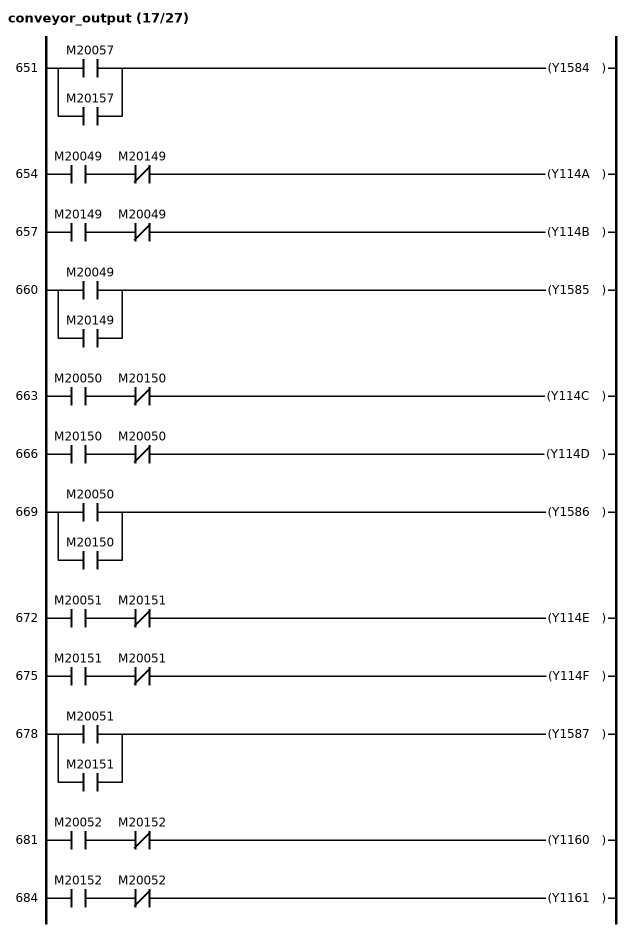
[picture p144: ladder of conveyor_output, rungs at steps 651 to 684]
651   LD      M20057
      OR      M20157
      OUT     Y1584
654   LD      M20049
      ANI     M20149
      OUT     Y114A
657   LD      M20149
      ANI     M20049
      OUT     Y114B
660   LD      M20049
      OR      M20149
      OUT     Y1585
663   LD      M20050
      ANI     M20150
      OUT     Y114C
666   LD      M20150
      ANI     M20050
      OUT     Y114D
669   LD      M20050
      OR      M20150
      OUT     Y1586
672   LD      M20051
      ANI     M20151
      OUT     Y114E
675   LD      M20151
      ANI     M20051
      OUT     Y114F
678   LD      M20051
      OR      M20151
      OUT     Y1587
681   LD      M20052
      ANI     M20152
      OUT     Y1160
684   LD      M20152
      ANI     M20052
      OUT     Y1161
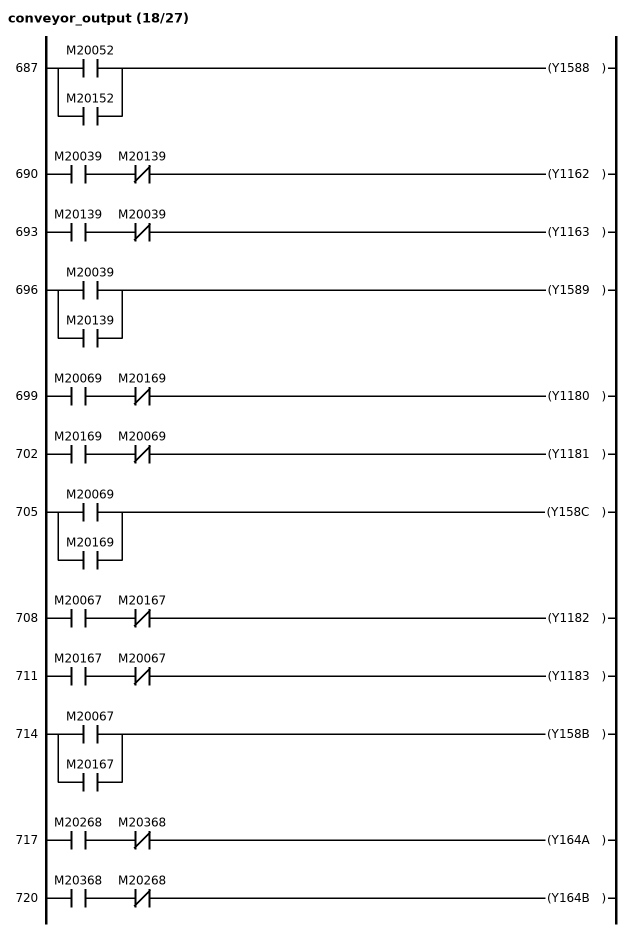
687   LD      M20052
      OR      M20152
      OUT     Y1588
690   LD      M20039
      ANI     M20139
      OUT     Y1162
693   LD      M20139
      ANI     M20039
      OUT     Y1163
696   LD      M20039
      OR      M20139
      OUT     Y1589
699   LD      M20069
      ANI     M20169
      OUT     Y1180
702   LD      M20169
      ANI     M20069
      OUT     Y1181
705   LD      M20069
      OR      M20169
      OUT     Y158C
708   LD      M20067
      ANI     M20167
      OUT     Y1182
711   LD      M20167
      ANI     M20067
      OUT     Y1183
714   LD      M20067
      OR      M20167
      OUT     Y158B
717   LD      M20268
      ANI     M20368
      OUT     Y164A
720   LD      M20368
      ANI     M20268
      OUT     Y164B
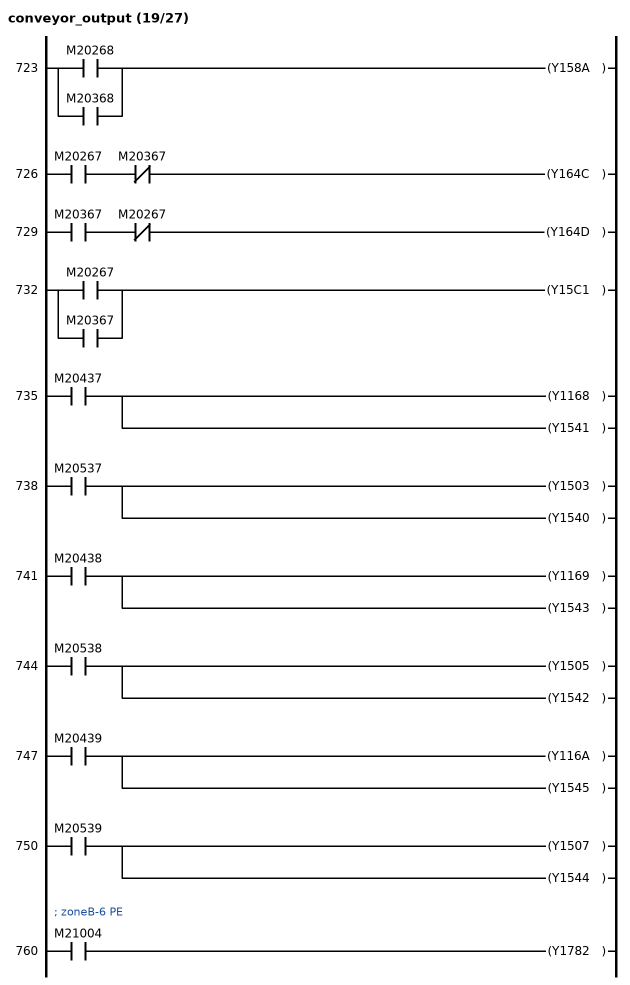
723   LD      M20268
      OR      M20368
      OUT     Y158A
726   LD      M20267
      ANI     M20367
      OUT     Y164C
729   LD      M20367
      ANI     M20267
      OUT     Y164D
732   LD      M20267
      OR      M20367
      OUT     Y15C1
735   LD      M20437
      OUT     Y1168
      OUT     Y1541
738   LD      M20537
      OUT     Y1503
      OUT     Y1540
741   LD      M20438
      OUT     Y1169
      OUT     Y1543
744   LD      M20538
      OUT     Y1505
      OUT     Y1542
747   LD      M20439
      OUT     Y116A
      OUT     Y1545
750   LD      M20539
      OUT     Y1507
      OUT     Y1544
; zoneB-6 PE
760   LD      M21004
      OUT     Y1782
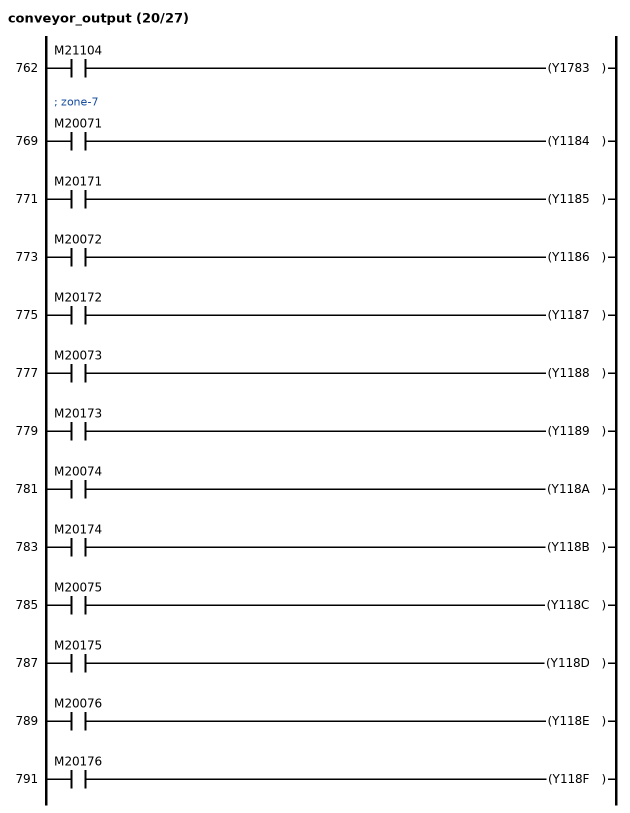
762   LD      M21104
      OUT     Y1783
; zone-7
769   LD      M20071
      OUT     Y1184
771   LD      M20171
      OUT     Y1185
773   LD      M20072
      OUT     Y1186
775   LD      M20172
      OUT     Y1187
777   LD      M20073
      OUT     Y1188
779   LD      M20173
      OUT     Y1189
781   LD      M20074
      OUT     Y118A
783   LD      M20174
      OUT     Y118B
785   LD      M20075
      OUT     Y118C
787   LD      M20175
      OUT     Y118D
789   LD      M20076
      OUT     Y118E
791   LD      M20176
      OUT     Y118F
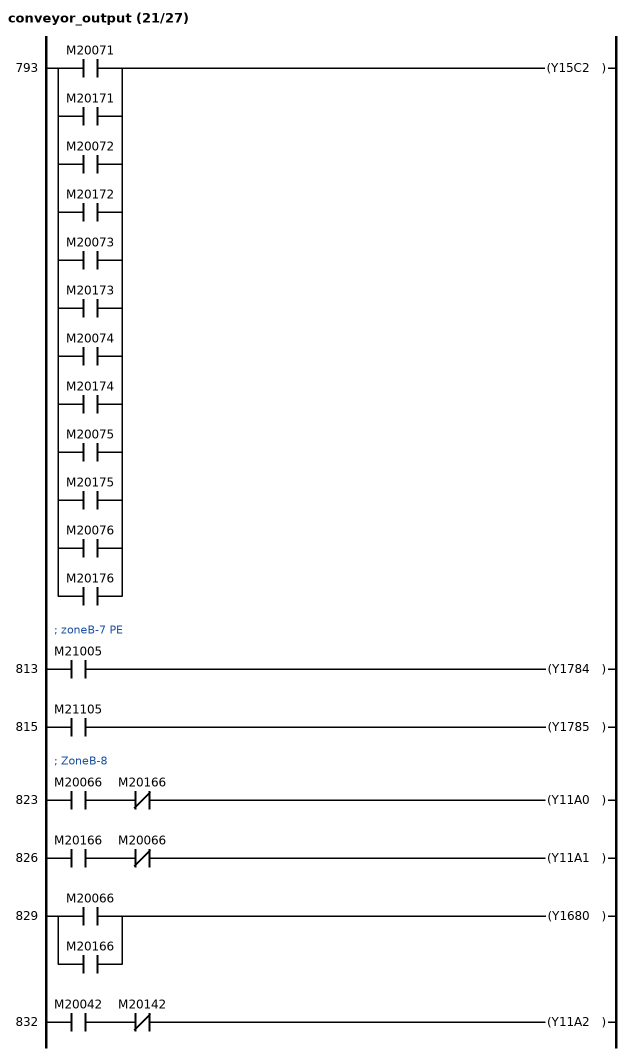
793   LD      M20071
      OR      M20171
      OR      M20072
      OR      M20172
      OR      M20073
      OR      M20173
      OR      M20074
      OR      M20174
      OR      M20075
      OR      M20175
      OR      M20076
      OR      M20176
      OUT     Y15C2
; zoneB-7 PE
813   LD      M21005
      OUT     Y1784
815   LD      M21105
      OUT     Y1785
; ZoneB-8
823   LD      M20066
      ANI     M20166
      OUT     Y11A0
826   LD      M20166
      ANI     M20066
      OUT     Y11A1
829   LD      M20066
      OR      M20166
      OUT     Y1680
832   LD      M20042
      ANI     M20142
      OUT     Y11A2
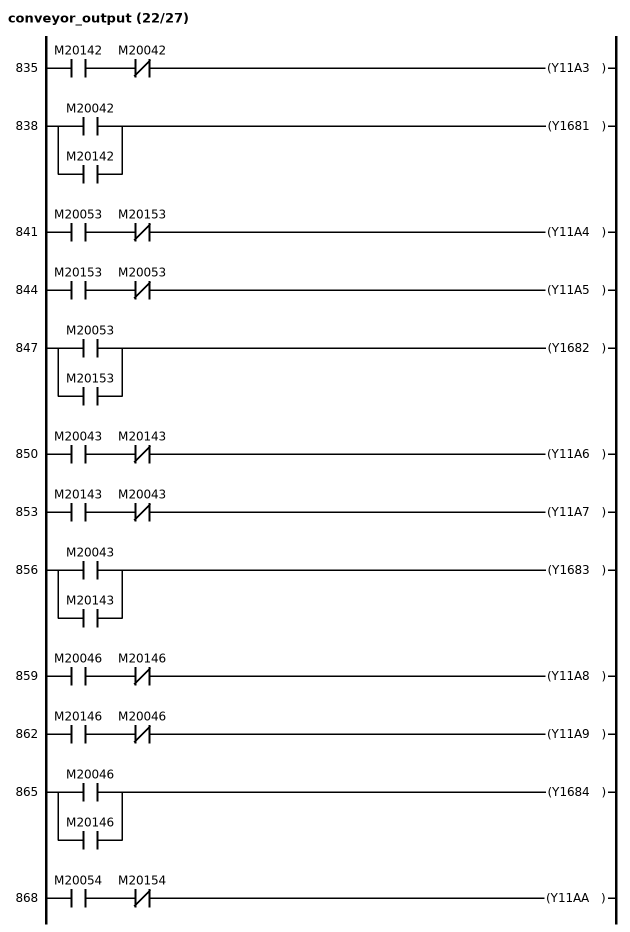
835   LD      M20142
      ANI     M20042
      OUT     Y11A3
838   LD      M20042
      OR      M20142
      OUT     Y1681
841   LD      M20053
      ANI     M20153
      OUT     Y11A4
844   LD      M20153
      ANI     M20053
      OUT     Y11A5
847   LD      M20053
      OR      M20153
      OUT     Y1682
850   LD      M20043
      ANI     M20143
      OUT     Y11A6
853   LD      M20143
      ANI     M20043
      OUT     Y11A7
856   LD      M20043
      OR      M20143
      OUT     Y1683
859   LD      M20046
      ANI     M20146
      OUT     Y11A8
862   LD      M20146
      ANI     M20046
      OUT     Y11A9
865   LD      M20046
      OR      M20146
      OUT     Y1684
868   LD      M20054
      ANI     M20154
      OUT     Y11AA
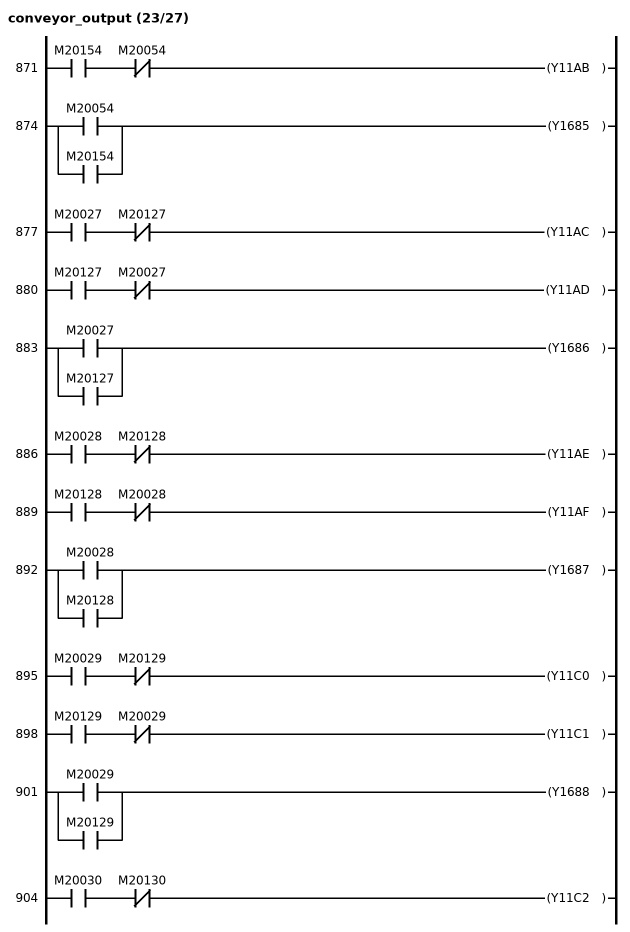
871   LD      M20154
      ANI     M20054
      OUT     Y11AB
874   LD      M20054
      OR      M20154
      OUT     Y1685
877   LD      M20027
      ANI     M20127
      OUT     Y11AC
880   LD      M20127
      ANI     M20027
      OUT     Y11AD
883   LD      M20027
      OR      M20127
      OUT     Y1686
886   LD      M20028
      ANI     M20128
      OUT     Y11AE
889   LD      M20128
      ANI     M20028
      OUT     Y11AF
892   LD      M20028
      OR      M20128
      OUT     Y1687
895   LD      M20029
      ANI     M20129
      OUT     Y11C0
898   LD      M20129
      ANI     M20029
      OUT     Y11C1
901   LD      M20029
      OR      M20129
      OUT     Y1688
904   LD      M20030
      ANI     M20130
      OUT     Y11C2
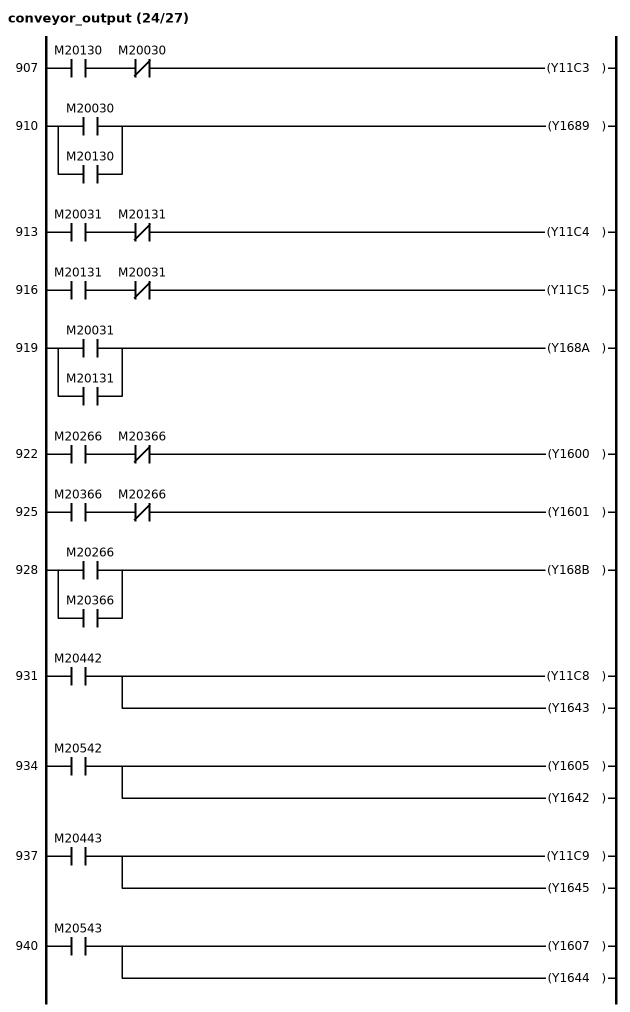
907   LD      M20130
      ANI     M20030
      OUT     Y11C3
910   LD      M20030
      OR      M20130
      OUT     Y1689
913   LD      M20031
      ANI     M20131
      OUT     Y11C4
916   LD      M20131
      ANI     M20031
      OUT     Y11C5
919   LD      M20031
      OR      M20131
      OUT     Y168A
922   LD      M20266
      ANI     M20366
      OUT     Y1600
925   LD      M20366
      ANI     M20266
      OUT     Y1601
928   LD      M20266
      OR      M20366
      OUT     Y168B
931   LD      M20442
      OUT     Y11C8
      OUT     Y1643
934   LD      M20542
      OUT     Y1605
      OUT     Y1642
937   LD      M20443
      OUT     Y11C9
      OUT     Y1645
940   LD      M20543
      OUT     Y1607
      OUT     Y1644
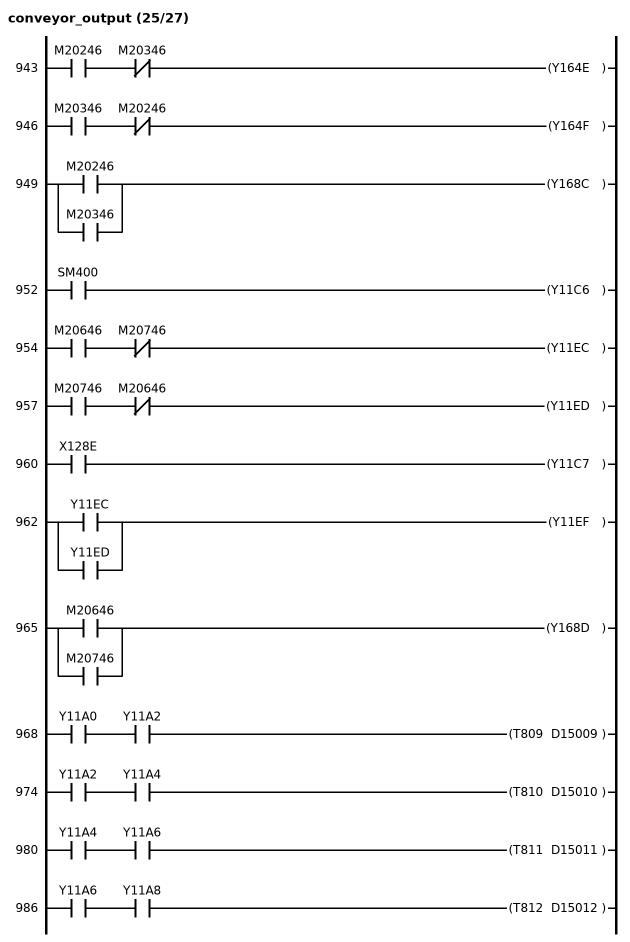
943   LD      M20246
      ANI     M20346
      OUT     Y164E
946   LD      M20346
      ANI     M20246
      OUT     Y164F
949   LD      M20246
      OR      M20346
      OUT     Y168C
952   LD      SM400
      OUT     Y11C6
954   LD      M20646
      ANI     M20746
      OUT     Y11EC
957   LD      M20746
      ANI     M20646
      OUT     Y11ED
960   LD      X128E
      OUT     Y11C7
962   LD      Y11EC
      OR      Y11ED
      OUT     Y11EF
965   LD      M20646
      OR      M20746
      OUT     Y168D
968   LD      Y11A0
      AND     Y11A2
      OUT     T809 D15009
974   LD      Y11A2
      AND     Y11A4
      OUT     T810 D15010
980   LD      Y11A4
      AND     Y11A6
      OUT     T811 D15011
986   LD      Y11A6
      AND     Y11A8
      OUT     T812 D15012
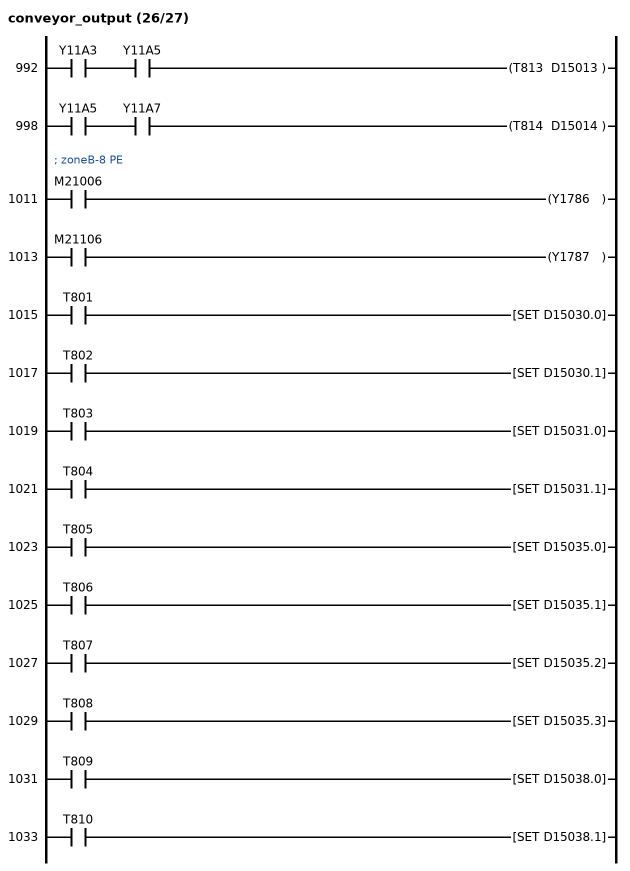
992   LD      Y11A3
      AND     Y11A5
      OUT     T813 D15013
998   LD      Y11A5
      AND     Y11A7
      OUT     T814 D15014
; zoneB-8 PE
1011  LD      M21006
      OUT     Y1786
1013  LD      M21106
      OUT     Y1787
1015  LD      T801
      SET     D15030.0
1017  LD      T802
      SET     D15030.1
1019  LD      T803
      SET     D15031.0
1021  LD      T804
      SET     D15031.1
1023  LD      T805
      SET     D15035.0
1025  LD      T806
      SET     D15035.1
1027  LD      T807
      SET     D15035.2
1029  LD      T808
      SET     D15035.3
1031  LD      T809
      SET     D15038.0
1033  LD      T810
      SET     D15038.1
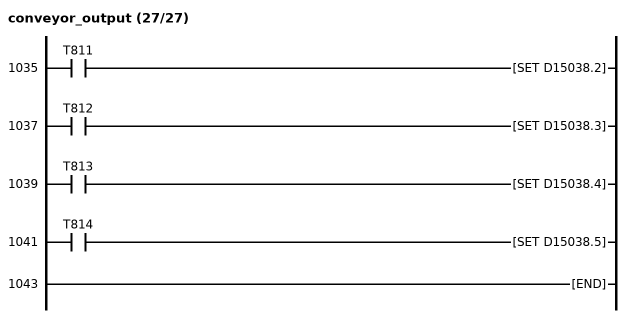
1035  LD      T811
      SET     D15038.2
1037  LD      T812
      SET     D15038.3
1039  LD      T813
      SET     D15038.4
1041  LD      T814
      SET     D15038.5
1043  END
END_PROGRAM

PROGRAM cover_system
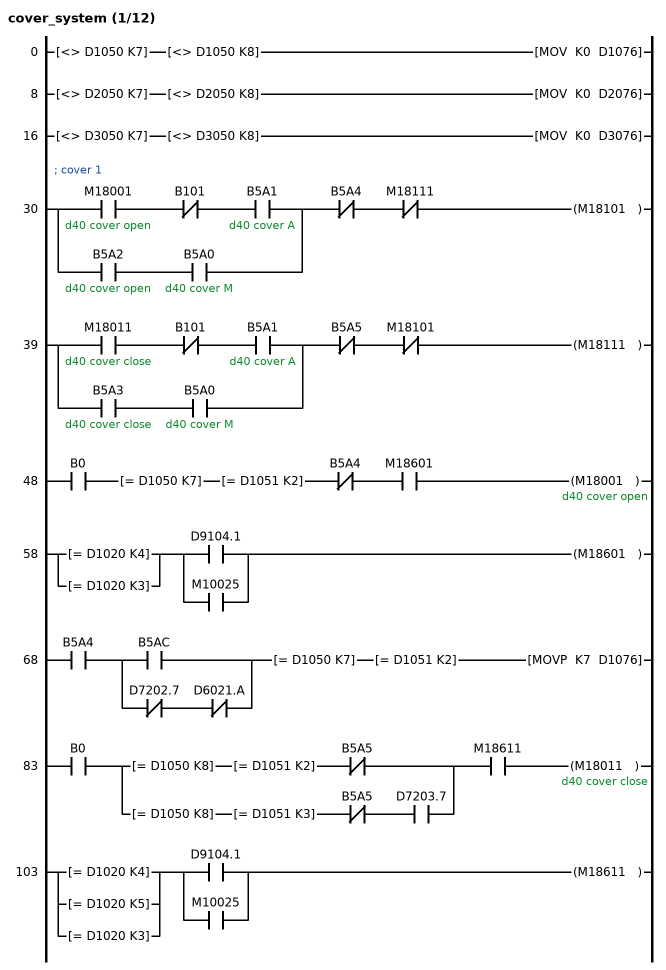
0     LD<>    D1050 K7
      AND<>   D1050 K8
      MOV     K0 D1076
8     LD<>    D2050 K7
      AND<>   D2050 K8
      MOV     K0 D2076
16    LD<>    D3050 K7
      AND<>   D3050 K8
      MOV     K0 D3076
; cover 1
30    LD      M18001  ; d40 cover open
      ANI     B101
      AND     B5A1  ; d40 cover A
      LD      B5A2  ; d40 cover open
      AND     B5A0  ; d40 cover M
      ORB
      ANI     B5A4
      ANI     M18111
      OUT     M18101
39    LD      M18011  ; d40 cover close
      ANI     B101
      AND     B5A1  ; d40 cover A
      LD      B5A3  ; d40 cover close
      AND     B5A0  ; d40 cover M
      ORB
      ANI     B5A5
      ANI     M18101
      OUT     M18111
48    LD      B0
      AND=    D1050 K7
      AND=    D1051 K2
      ANI     B5A4
      AND     M18601
      OUT     M18001  ; d40 cover open
58    LD=     D1020 K4
      OR=     D1020 K3
      LD      D9104.1
      OR      M10025
      ANB
      OUT     M18601
68    LD      B5A4
      LD      B5AC
      LDI     D7202.7
      ANI     D6021.A
      ORB
      ANB
      AND=    D1050 K7
      AND=    D1051 K2
      MOVP    K7 D1076
83    LD      B0
      LD=     D1050 K8
      AND=    D1051 K2
      ANI     B5A5
      LD=     D1050 K8
      AND=    D1051 K3
      ANI     B5A5
      AND     D7203.7
      ORB
      ANB
      AND     M18611
      OUT     M18011  ; d40 cover close
103   LD=     D1020 K4
      OR=     D1020 K5
      OR=     D1020 K3
      LD      D9104.1
      OR      M10025
      ANB
      OUT     M18611
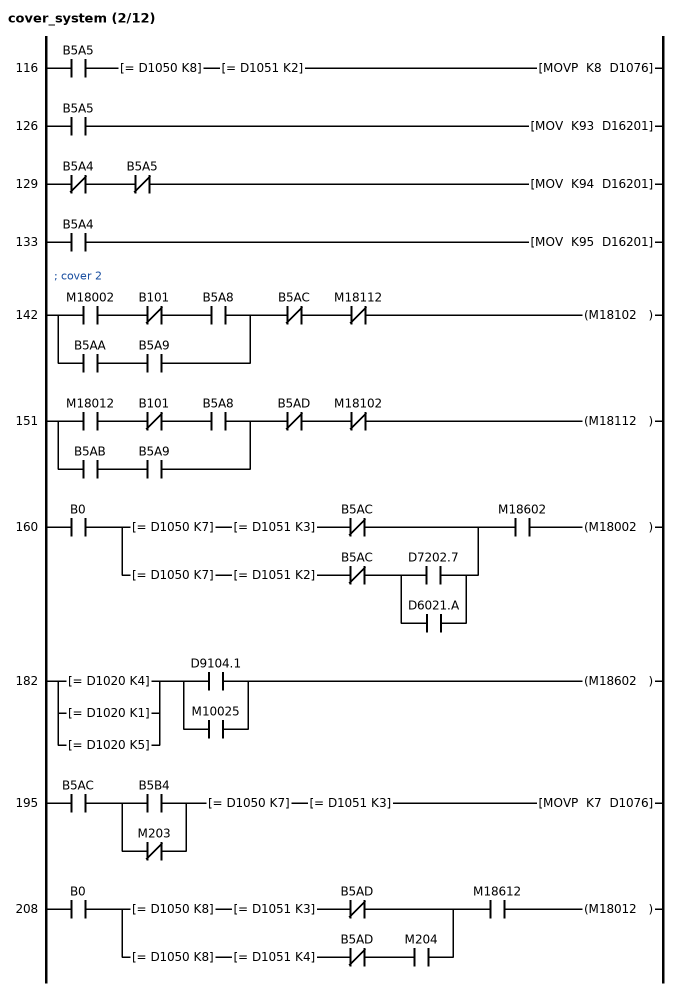
116   LD      B5A5
      AND=    D1050 K8
      AND=    D1051 K2
      MOVP    K8 D1076
126   LD      B5A5
      MOV     K93 D16201
129   LDI     B5A4
      ANI     B5A5
      MOV     K94 D16201
133   LD      B5A4
      MOV     K95 D16201
; cover 2
142   LD      M18002
      ANI     B101
      AND     B5A8
      LD      B5AA
      AND     B5A9
      ORB
      ANI     B5AC
      ANI     M18112
      OUT     M18102
151   LD      M18012
      ANI     B101
      AND     B5A8
      LD      B5AB
      AND     B5A9
      ORB
      ANI     B5AD
      ANI     M18102
      OUT     M18112
160   LD      B0
      LD=     D1050 K7
      AND=    D1051 K3
      ANI     B5AC
      LD=     D1050 K7
      AND=    D1051 K2
      ANI     B5AC
      LD      D7202.7
      OR      D6021.A
      ANB
      ORB
      ANB
      AND     M18602
      OUT     M18002
182   LD=     D1020 K4
      OR=     D1020 K1
      OR=     D1020 K5
      LD      D9104.1
      OR      M10025
      ANB
      OUT     M18602
195   LD      B5AC
      LD      B5B4
      ORI     M203
      ANB
      AND=    D1050 K7
      AND=    D1051 K3
      MOVP    K7 D1076
208   LD      B0
      LD=     D1050 K8
      AND=    D1051 K3
      ANI     B5AD
      LD=     D1050 K8
      AND=    D1051 K4
      ANI     B5AD
      AND     M204
      ORB
      ANB
      AND     M18612
      OUT     M18012
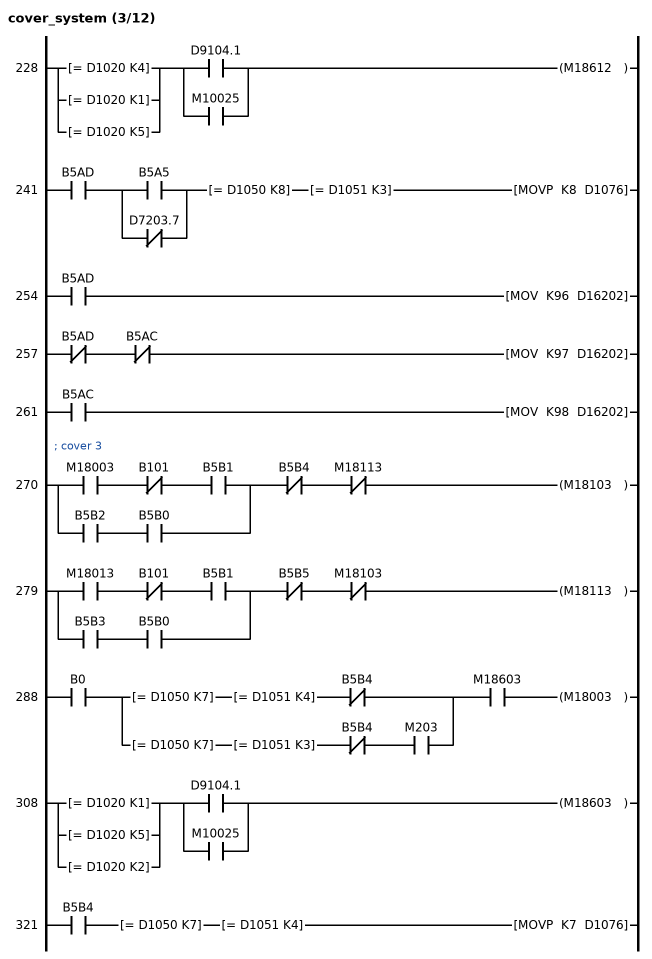
228   LD=     D1020 K4
      OR=     D1020 K1
      OR=     D1020 K5
      LD      D9104.1
      OR      M10025
      ANB
      OUT     M18612
241   LD      B5AD
      LD      B5A5
      ORI     D7203.7
      ANB
      AND=    D1050 K8
      AND=    D1051 K3
      MOVP    K8 D1076
254   LD      B5AD
      MOV     K96 D16202
257   LDI     B5AD
      ANI     B5AC
      MOV     K97 D16202
261   LD      B5AC
      MOV     K98 D16202
; cover 3
270   LD      M18003
      ANI     B101
      AND     B5B1
      LD      B5B2
      AND     B5B0
      ORB
      ANI     B5B4
      ANI     M18113
      OUT     M18103
279   LD      M18013
      ANI     B101
      AND     B5B1
      LD      B5B3
      AND     B5B0
      ORB
      ANI     B5B5
      ANI     M18103
      OUT     M18113
288   LD      B0
      LD=     D1050 K7
      AND=    D1051 K4
      ANI     B5B4
      LD=     D1050 K7
      AND=    D1051 K3
      ANI     B5B4
      AND     M203
      ORB
      ANB
      AND     M18603
      OUT     M18003
308   LD=     D1020 K1
      OR=     D1020 K5
      OR=     D1020 K2
      LD      D9104.1
      OR      M10025
      ANB
      OUT     M18603
321   LD      B5B4
      AND=    D1050 K7
      AND=    D1051 K4
      MOVP    K7 D1076
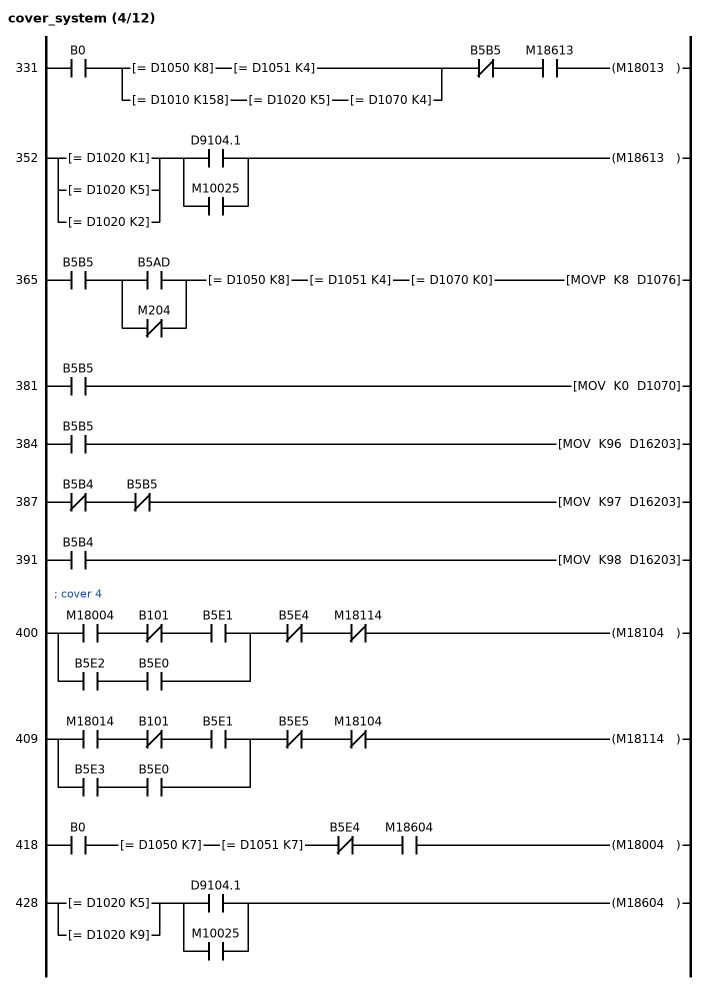
331   LD      B0
      LD=     D1050 K8
      AND=    D1051 K4
      LD=     D1010 K158
      AND=    D1020 K5
      AND=    D1070 K4
      ORB
      ANB
      ANI     B5B5
      AND     M18613
      OUT     M18013
352   LD=     D1020 K1
      OR=     D1020 K5
      OR=     D1020 K2
      LD      D9104.1
      OR      M10025
      ANB
      OUT     M18613
365   LD      B5B5
      LD      B5AD
      ORI     M204
      ANB
      AND=    D1050 K8
      AND=    D1051 K4
      AND=    D1070 K0
      MOVP    K8 D1076
381   LD      B5B5
      MOV     K0 D1070
384   LD      B5B5
      MOV     K96 D16203
387   LDI     B5B4
      ANI     B5B5
      MOV     K97 D16203
391   LD      B5B4
      MOV     K98 D16203
; cover 4
400   LD      M18004
      ANI     B101
      AND     B5E1
      LD      B5E2
      AND     B5E0
      ORB
      ANI     B5E4
      ANI     M18114
      OUT     M18104
409   LD      M18014
      ANI     B101
      AND     B5E1
      LD      B5E3
      AND     B5E0
      ORB
      ANI     B5E5
      ANI     M18104
      OUT     M18114
418   LD      B0
      AND=    D1050 K7
      AND=    D1051 K7
      ANI     B5E4
      AND     M18604
      OUT     M18004
428   LD=     D1020 K5
      OR=     D1020 K9
      LD      D9104.1
      OR      M10025
      ANB
      OUT     M18604
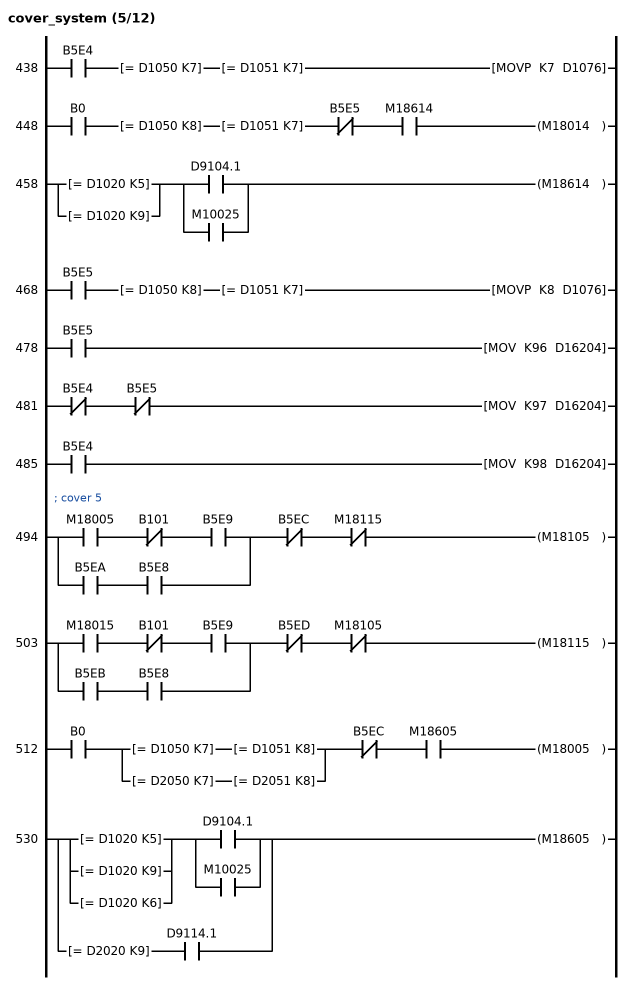
438   LD      B5E4
      AND=    D1050 K7
      AND=    D1051 K7
      MOVP    K7 D1076
448   LD      B0
      AND=    D1050 K8
      AND=    D1051 K7
      ANI     B5E5
      AND     M18614
      OUT     M18014
458   LD=     D1020 K5
      OR=     D1020 K9
      LD      D9104.1
      OR      M10025
      ANB
      OUT     M18614
468   LD      B5E5
      AND=    D1050 K8
      AND=    D1051 K7
      MOVP    K8 D1076
478   LD      B5E5
      MOV     K96 D16204
481   LDI     B5E4
      ANI     B5E5
      MOV     K97 D16204
485   LD      B5E4
      MOV     K98 D16204
; cover 5
494   LD      M18005
      ANI     B101
      AND     B5E9
      LD      B5EA
      AND     B5E8
      ORB
      ANI     B5EC
      ANI     M18115
      OUT     M18105
503   LD      M18015
      ANI     B101
      AND     B5E9
      LD      B5EB
      AND     B5E8
      ORB
      ANI     B5ED
      ANI     M18105
      OUT     M18115
512   LD      B0
      LD=     D1050 K7
      AND=    D1051 K8
      LD=     D2050 K7
      AND=    D2051 K8
      ORB
      ANB
      ANI     B5EC
      AND     M18605
      OUT     M18005
530   LD=     D1020 K5
      OR=     D1020 K9
      OR=     D1020 K6
      LD      D9104.1
      OR      M10025
      ANB
      LD=     D2020 K9
      AND     D9114.1
      ORB
      OUT     M18605
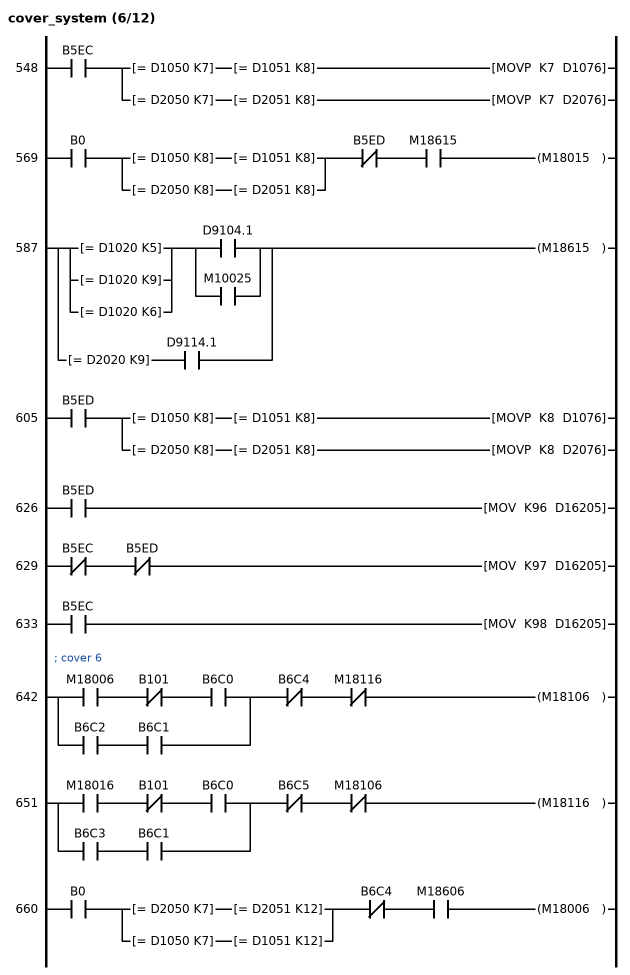
548   LD      B5EC
      MPS
      AND=    D1050 K7
      AND=    D1051 K8
      MOVP    K7 D1076
      MPP
      AND=    D2050 K7
      AND=    D2051 K8
      MOVP    K7 D2076
569   LD      B0
      LD=     D1050 K8
      AND=    D1051 K8
      LD=     D2050 K8
      AND=    D2051 K8
      ORB
      ANB
      ANI     B5ED
      AND     M18615
      OUT     M18015
587   LD=     D1020 K5
      OR=     D1020 K9
      OR=     D1020 K6
      LD      D9104.1
      OR      M10025
      ANB
      LD=     D2020 K9
      AND     D9114.1
      ORB
      OUT     M18615
605   LD      B5ED
      MPS
      AND=    D1050 K8
      AND=    D1051 K8
      MOVP    K8 D1076
      MPP
      AND=    D2050 K8
      AND=    D2051 K8
      MOVP    K8 D2076
626   LD      B5ED
      MOV     K96 D16205
629   LDI     B5EC
      ANI     B5ED
      MOV     K97 D16205
633   LD      B5EC
      MOV     K98 D16205
; cover 6
642   LD      M18006
      ANI     B101
      AND     B6C0
      LD      B6C2
      AND     B6C1
      ORB
      ANI     B6C4
      ANI     M18116
      OUT     M18106
651   LD      M18016
      ANI     B101
      AND     B6C0
      LD      B6C3
      AND     B6C1
      ORB
      ANI     B6C5
      ANI     M18106
      OUT     M18116
660   LD      B0
      LD=     D2050 K7
      AND=    D2051 K12
      LD=     D1050 K7
      AND=    D1051 K12
      ORB
      ANB
      ANI     B6C4
      AND     M18606
      OUT     M18006
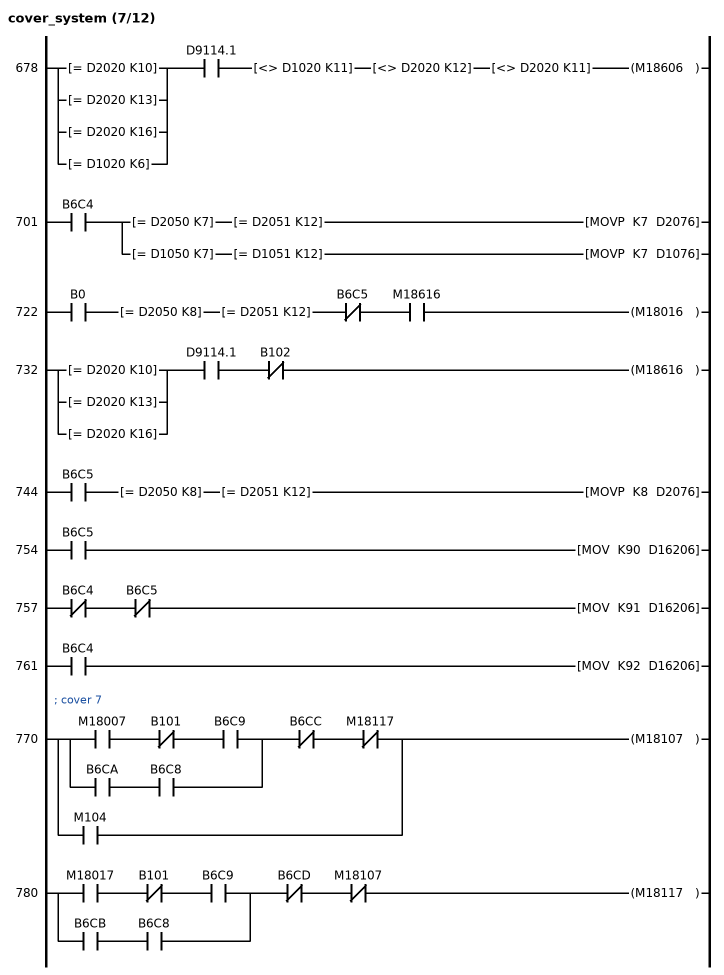
678   LD=     D2020 K10
      OR=     D2020 K13
      OR=     D2020 K16
      OR=     D1020 K6
      AND     D9114.1
      AND<>   D1020 K11
      AND<>   D2020 K12
      AND<>   D2020 K11
      OUT     M18606
701   LD      B6C4
      MPS
      AND=    D2050 K7
      AND=    D2051 K12
      MOVP    K7 D2076
      MPP
      AND=    D1050 K7
      AND=    D1051 K12
      MOVP    K7 D1076
722   LD      B0
      AND=    D2050 K8
      AND=    D2051 K12
      ANI     B6C5
      AND     M18616
      OUT     M18016
732   LD=     D2020 K10
      OR=     D2020 K13
      OR=     D2020 K16
      AND     D9114.1
      ANI     B102
      OUT     M18616
744   LD      B6C5
      AND=    D2050 K8
      AND=    D2051 K12
      MOVP    K8 D2076
754   LD      B6C5
      MOV     K90 D16206
757   LDI     B6C4
      ANI     B6C5
      MOV     K91 D16206
761   LD      B6C4
      MOV     K92 D16206
; cover 7
770   LD      M18007
      ANI     B101
      AND     B6C9
      LD      B6CA
      AND     B6C8
      ORB
      ANI     B6CC
      ANI     M18117
      OR      M104
      OUT     M18107
780   LD      M18017
      ANI     B101
      AND     B6C9
      LD      B6CB
      AND     B6C8
      ORB
      ANI     B6CD
      ANI     M18107
      OUT     M18117
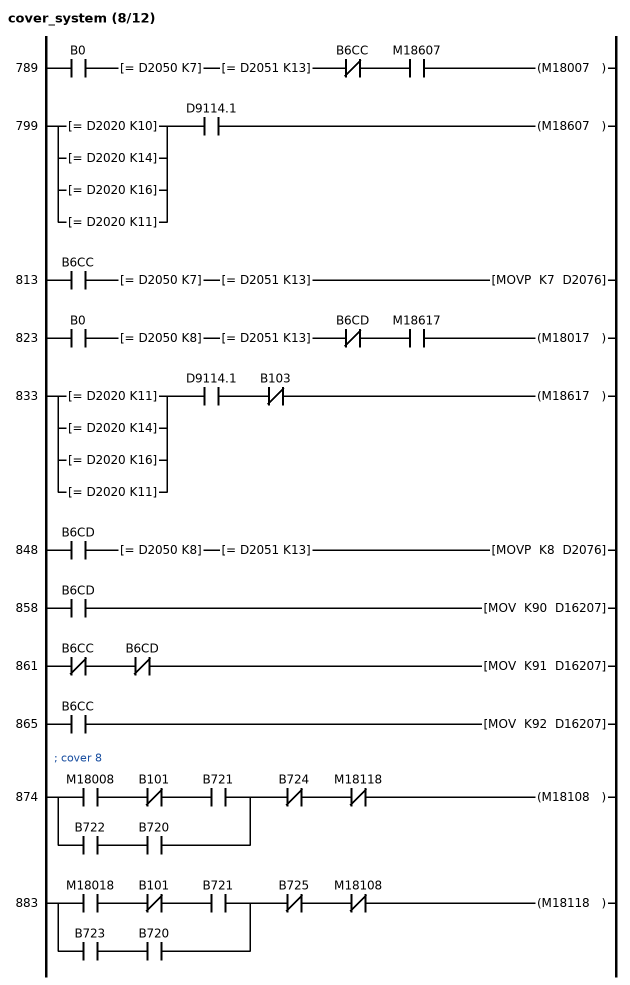
789   LD      B0
      AND=    D2050 K7
      AND=    D2051 K13
      ANI     B6CC
      AND     M18607
      OUT     M18007
799   LD=     D2020 K10
      OR=     D2020 K14
      OR=     D2020 K16
      OR=     D2020 K11
      AND     D9114.1
      OUT     M18607
813   LD      B6CC
      AND=    D2050 K7
      AND=    D2051 K13
      MOVP    K7 D2076
823   LD      B0
      AND=    D2050 K8
      AND=    D2051 K13
      ANI     B6CD
      AND     M18617
      OUT     M18017
833   LD=     D2020 K11
      OR=     D2020 K14
      OR=     D2020 K16
      OR=     D2020 K11
      AND     D9114.1
      ANI     B103
      OUT     M18617
848   LD      B6CD
      AND=    D2050 K8
      AND=    D2051 K13
      MOVP    K8 D2076
858   LD      B6CD
      MOV     K90 D16207
861   LDI     B6CC
      ANI     B6CD
      MOV     K91 D16207
865   LD      B6CC
      MOV     K92 D16207
; cover 8
874   LD      M18008
      ANI     B101
      AND     B721
      LD      B722
      AND     B720
      ORB
      ANI     B724
      ANI     M18118
      OUT     M18108
883   LD      M18018
      ANI     B101
      AND     B721
      LD      B723
      AND     B720
      ORB
      ANI     B725
      ANI     M18108
      OUT     M18118
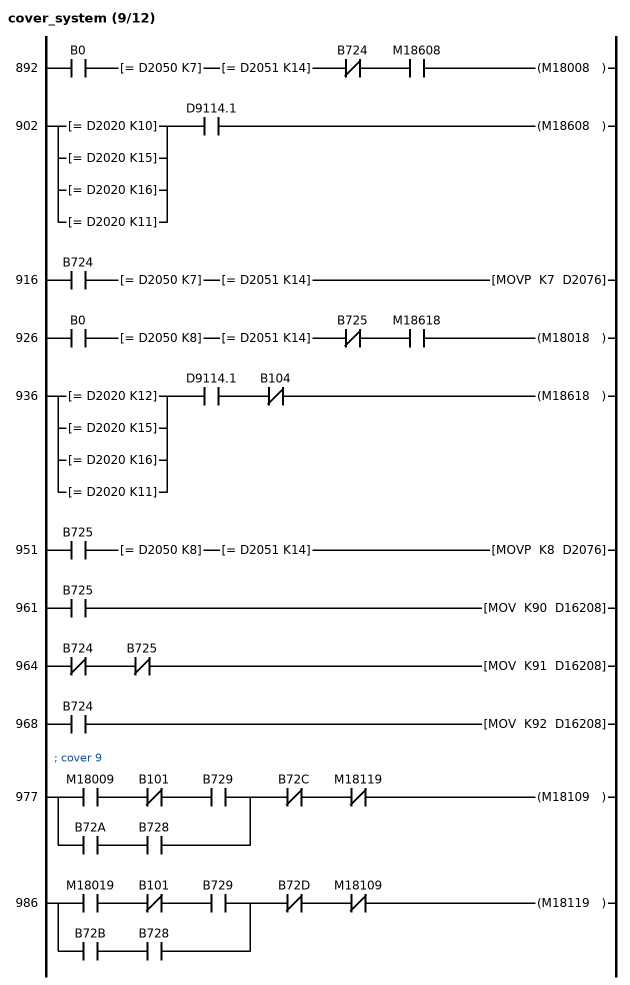
892   LD      B0
      AND=    D2050 K7
      AND=    D2051 K14
      ANI     B724
      AND     M18608
      OUT     M18008
902   LD=     D2020 K10
      OR=     D2020 K15
      OR=     D2020 K16
      OR=     D2020 K11
      AND     D9114.1
      OUT     M18608
916   LD      B724
      AND=    D2050 K7
      AND=    D2051 K14
      MOVP    K7 D2076
926   LD      B0
      AND=    D2050 K8
      AND=    D2051 K14
      ANI     B725
      AND     M18618
      OUT     M18018
936   LD=     D2020 K12
      OR=     D2020 K15
      OR=     D2020 K16
      OR=     D2020 K11
      AND     D9114.1
      ANI     B104
      OUT     M18618
951   LD      B725
      AND=    D2050 K8
      AND=    D2051 K14
      MOVP    K8 D2076
961   LD      B725
      MOV     K90 D16208
964   LDI     B724
      ANI     B725
      MOV     K91 D16208
968   LD      B724
      MOV     K92 D16208
; cover 9
977   LD      M18009
      ANI     B101
      AND     B729
      LD      B72A
      AND     B728
      ORB
      ANI     B72C
      ANI     M18119
      OUT     M18109
986   LD      M18019
      ANI     B101
      AND     B729
      LD      B72B
      AND     B728
      ORB
      ANI     B72D
      ANI     M18109
      OUT     M18119
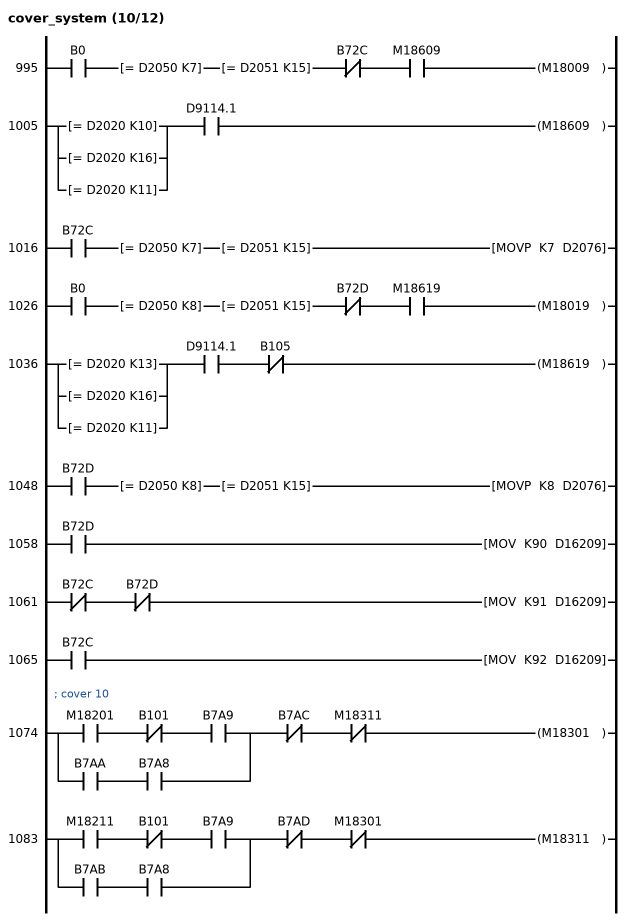
995   LD      B0
      AND=    D2050 K7
      AND=    D2051 K15
      ANI     B72C
      AND     M18609
      OUT     M18009
1005  LD=     D2020 K10
      OR=     D2020 K16
      OR=     D2020 K11
      AND     D9114.1
      OUT     M18609
1016  LD      B72C
      AND=    D2050 K7
      AND=    D2051 K15
      MOVP    K7 D2076
1026  LD      B0
      AND=    D2050 K8
      AND=    D2051 K15
      ANI     B72D
      AND     M18619
      OUT     M18019
1036  LD=     D2020 K13
      OR=     D2020 K16
      OR=     D2020 K11
      AND     D9114.1
      ANI     B105
      OUT     M18619
1048  LD      B72D
      AND=    D2050 K8
      AND=    D2051 K15
      MOVP    K8 D2076
1058  LD      B72D
      MOV     K90 D16209
1061  LDI     B72C
      ANI     B72D
      MOV     K91 D16209
1065  LD      B72C
      MOV     K92 D16209
; cover 10
1074  LD      M18201
      ANI     B101
      AND     B7A9
      LD      B7AA
      AND     B7A8
      ORB
      ANI     B7AC
      ANI     M18311
      OUT     M18301
1083  LD      M18211
      ANI     B101
      AND     B7A9
      LD      B7AB
      AND     B7A8
      ORB
      ANI     B7AD
      ANI     M18301
      OUT     M18311
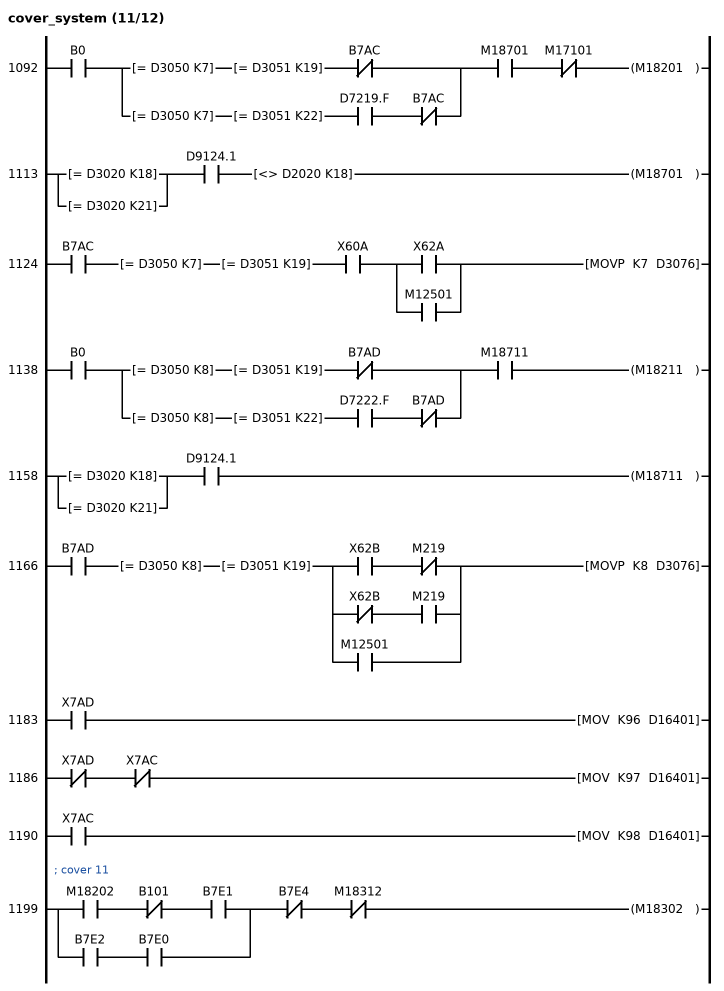
1092  LD      B0
      LD=     D3050 K7
      AND=    D3051 K19
      ANI     B7AC
      LD=     D3050 K7
      AND=    D3051 K22
      AND     D7219.F
      ANI     B7AC
      ORB
      ANB
      AND     M18701
      ANI     M17101
      OUT     M18201
1113  LD=     D3020 K18
      OR=     D3020 K21
      AND     D9124.1
      AND<>   D2020 K18
      OUT     M18701
1124  LD      B7AC
      AND=    D3050 K7
      AND=    D3051 K19
      AND     X60A
      LD      X62A
      OR      M12501
      ANB
      MOVP    K7 D3076
1138  LD      B0
      LD=     D3050 K8
      AND=    D3051 K19
      ANI     B7AD
      LD=     D3050 K8
      AND=    D3051 K22
      AND     D7222.F
      ANI     B7AD
      ORB
      ANB
      AND     M18711
      OUT     M18211
1158  LD=     D3020 K18
      OR=     D3020 K21
      AND     D9124.1
      OUT     M18711
1166  LD      B7AD
      AND=    D3050 K8
      AND=    D3051 K19
      LD      X62B
      ANI     M219
      LDI     X62B
      AND     M219
      ORB
      OR      M12501
      ANB
      MOVP    K8 D3076
1183  LD      X7AD
      MOV     K96 D16401
1186  LDI     X7AD
      ANI     X7AC
      MOV     K97 D16401
1190  LD      X7AC
      MOV     K98 D16401
; cover 11
1199  LD      M18202
      ANI     B101
      AND     B7E1
      LD      B7E2
      AND     B7E0
      ORB
      ANI     B7E4
      ANI     M18312
      OUT     M18302
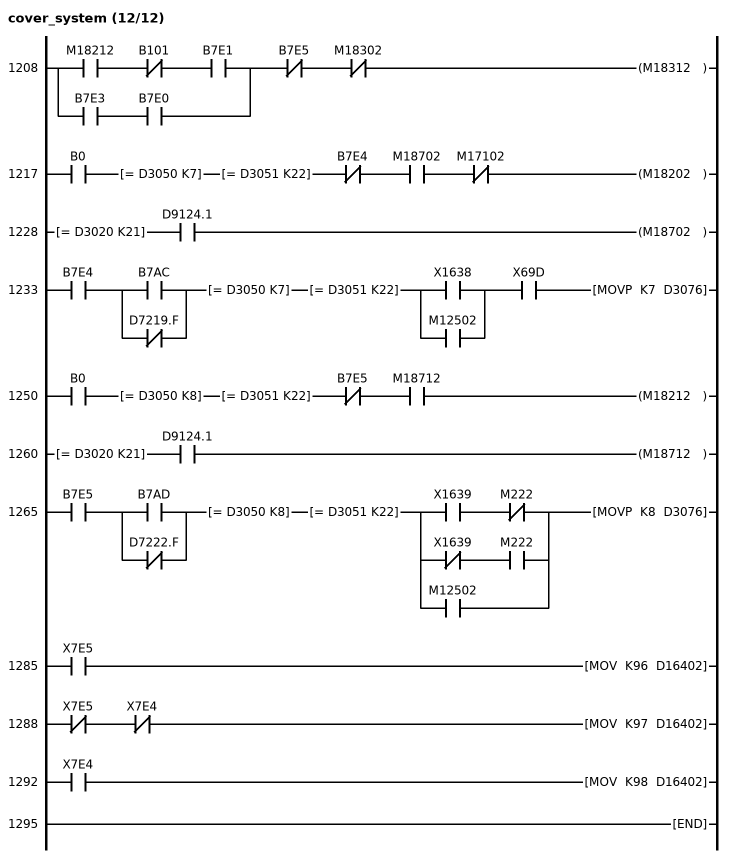
1208  LD      M18212
      ANI     B101
      AND     B7E1
      LD      B7E3
      AND     B7E0
      ORB
      ANI     B7E5
      ANI     M18302
      OUT     M18312
1217  LD      B0
      AND=    D3050 K7
      AND=    D3051 K22
      ANI     B7E4
      AND     M18702
      ANI     M17102
      OUT     M18202
1228  LD=     D3020 K21
      AND     D9124.1
      OUT     M18702
1233  LD      B7E4
      LD      B7AC
      ORI     D7219.F
      ANB
      AND=    D3050 K7
      AND=    D3051 K22
      LD      X1638
      OR      M12502
      ANB
      AND     X69D
      MOVP    K7 D3076
1250  LD      B0
      AND=    D3050 K8
      AND=    D3051 K22
      ANI     B7E5
      AND     M18712
      OUT     M18212
1260  LD=     D3020 K21
      AND     D9124.1
      OUT     M18712
1265  LD      B7E5
      LD      B7AD
      ORI     D7222.F
      ANB
      AND=    D3050 K8
      AND=    D3051 K22
      LD      X1639
      ANI     M222
      LDI     X1639
      AND     M222
      ORB
      OR      M12502
      ANB
      MOVP    K8 D3076
1285  LD      X7E5
      MOV     K96 D16402
1288  LDI     X7E5
      ANI     X7E4
      MOV     K97 D16402
1292  LD      X7E4
      MOV     K98 D16402
1295  END
END_PROGRAM

PROGRAM coveyor_system
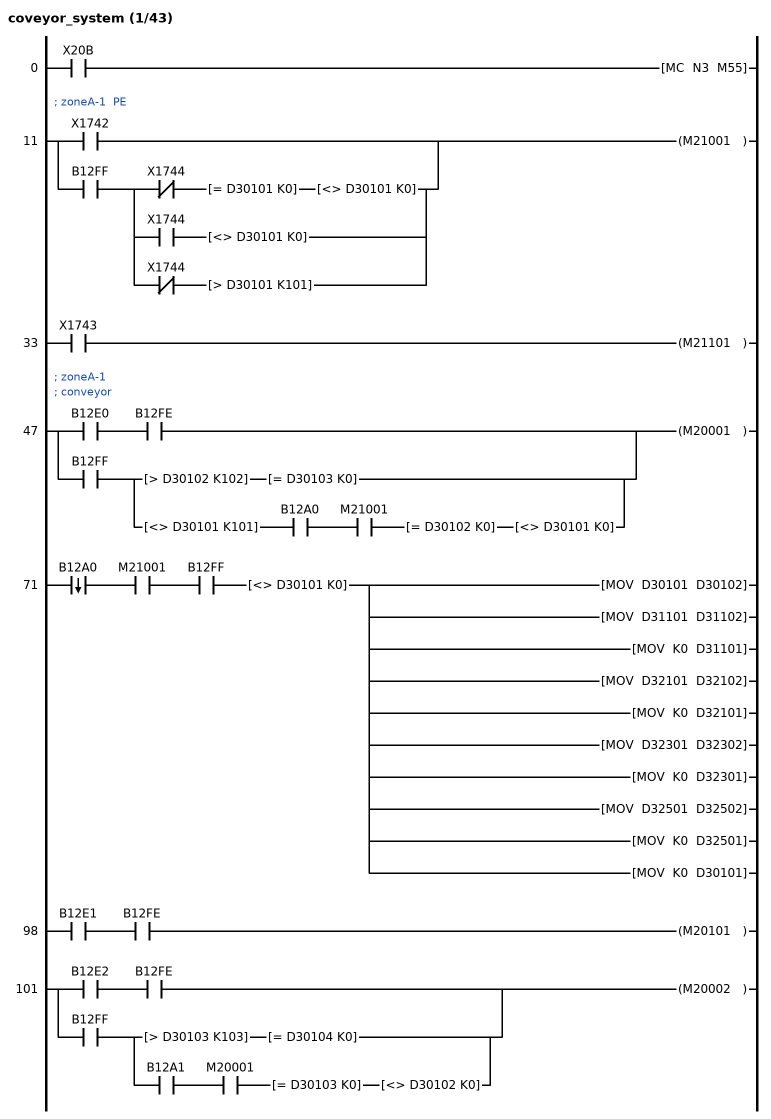
0     LD      X20B
      MC      N3 M55
; zoneA-1  PE
11    LD      X1742
      LD      B12FF
      LDI     X1744
      AND=    D30101 K0
      AND<>   D30101 K0
      LD      X1744
      AND<>   D30101 K0
      ORB
      LDI     X1744
      AND>    D30101 K101
      ORB
      ANB
      ORB
      OUT     M21001
33    LD      X1743
      OUT     M21101
; zoneA-1
; conveyor
47    LD      B12E0
      AND     B12FE
      LD      B12FF
      LD>     D30102 K102
      AND=    D30103 K0
      LD<>    D30101 K101
      AND     B12A0
      AND     M21001
      AND=    D30102 K0
      AND<>   D30101 K0
      ORB
      ANB
      ORB
      OUT     M20001
71    LDF     B12A0
      AND     M21001
      AND     B12FF
      AND<>   D30101 K0
      MOV     D30101 D30102
      MOV     D31101 D31102
      MOV     K0 D31101
      MOV     D32101 D32102
      MOV     K0 D32101
      MOV     D32301 D32302
      MOV     K0 D32301
      MOV     D32501 D32502
      MOV     K0 D32501
      MOV     K0 D30101
98    LD      B12E1
      AND     B12FE
      OUT     M20101
101   LD      B12E2
      AND     B12FE
      LD      B12FF
      LD>     D30103 K103
      AND=    D30104 K0
      LD      B12A1
      AND     M20001
      AND=    D30103 K0
      AND<>   D30102 K0
      ORB
      ANB
      ORB
      OUT     M20002
